{attribute 'hide_all_locals'}
{attribute 'enable_dynamic_creation'}
FUNCTION_BLOCK BoolBindingReadOnly IMPLEMENTS BoolBindable
VAR
	ref : REFERENCE TO BOOL;
	_Negate : BOOL;
END_VAR

METHOD Bind
VAR_INPUT
	boolean : REFERENCE TO BOOL;
END_VAR
ref REF= boolean;
END_METHOD

{attribute 'monitoring' := 'call'}
PROPERTY IsBinded : BOOL
GET
IsBinded := __ISVALIDREF(ref);
END_GET
END_PROPERTY

PROPERTY Negate : BOOL
GET
Negate := _Negate;
END_GET
SET
_Negate := Negate;
END_SET
END_PROPERTY

{attribute 'monitoring' := 'call'}
PROPERTY Value : BOOL
GET
Value := ref XOR _Negate;
END_GET
END_PROPERTY

END_FUNCTION_BLOCK

(* stored: Version 1.1.0.1
   POU BoolBindingReadOnly: Id {f035c595-f3d7-4302-a6a4-0e368016167c}, SpecialFunc None
   Method Bind: Id {e983f9b6-0ab6-437c-96e5-a762d13ac396}
   Property IsBinded: Id {b98b2f4c-bef9-4cbe-8145-c6052f4c6749}
   Get Get: Id {c3ecef46-ab78-4488-800b-ef0c98e1f08e}
   Property Negate: Id {71f8018d-5674-4339-86f2-5a523bdef0bb}
   Get Get: Id {5f5839d5-85dd-4f15-9ce5-a576769aa98b}
   Set Set: Id {28879c35-1f76-4604-9898-7f1bf0b41a79}
   Property Value: Id {be34ded7-c52a-40b6-be7d-89514242f0d3}
   Get Get: Id {c9cb8b85-06e5-474e-ad80-b0bc709ea14b} *)
